FUNCTION_BLOCK bfb_offpeak_charging
  (* Standard: 61499-2 *)
  (* Version 0.1, 2018-00-09, palme, DESKTOP-TGOEKBD *)
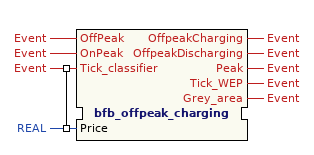
  EVENT_INPUT
    OffPeak;
    OnPeak;
    Tick_classifier WITH Price;
  END_EVENT
  EVENT_OUTPUT
    OffpeakCharging;
    OffpeakDischarging;
    Peak;
    Tick_WEP;
    Grey_area;
  END_EVENT
  VAR_INPUT
    Price : REAL;
  END_VAR
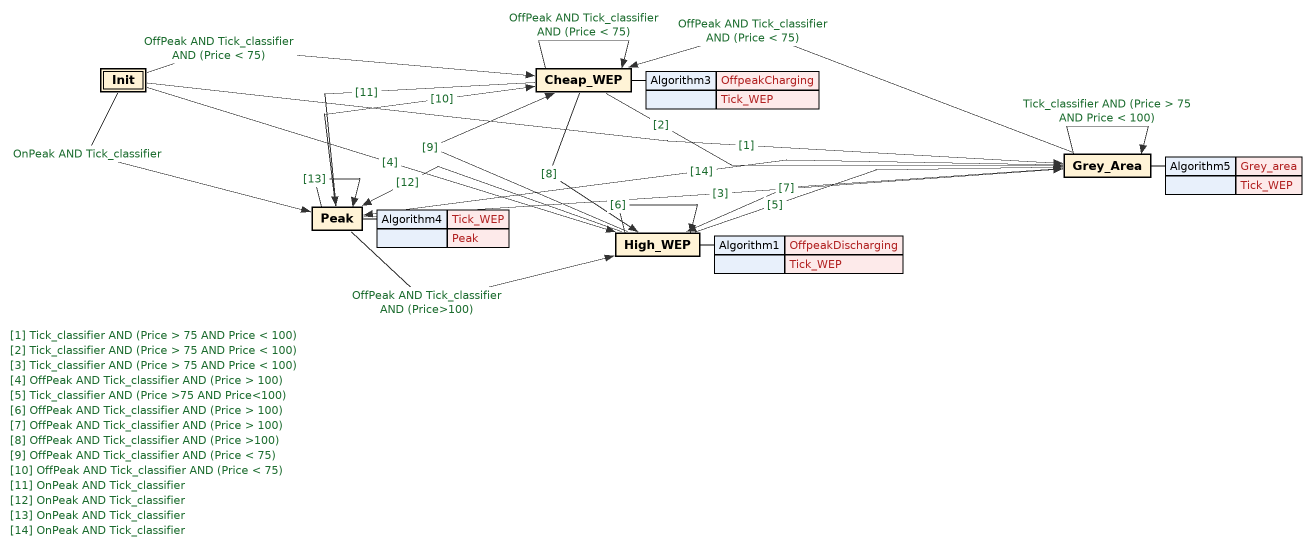
  EC_STATES
    Init;
    Cheap_WEP : Algorithm3 -> OffpeakCharging, -> Tick_WEP;
    High_WEP : Algorithm1 -> OffpeakDischarging, -> Tick_WEP;
    Peak : Algorithm4 -> Tick_WEP, -> Peak;
    Grey_Area : Algorithm5 -> Grey_area, -> Tick_WEP;
  END_STATES
  EC_TRANSITIONS
    Init TO Peak := OnPeak AND Tick_classifier;
    Init TO Grey_Area := Tick_classifier AND (Price > 75 AND Price < 100);
    Init TO Cheap_WEP := OffPeak AND Tick_classifier AND (Price < 75);
    Init TO High_WEP := OffPeak AND Tick_classifier AND (Price > 100);
    Cheap_WEP TO Peak := OnPeak AND Tick_classifier;
    Cheap_WEP TO Grey_Area := Tick_classifier AND (Price > 75 AND Price < 100);
    Cheap_WEP TO High_WEP := OffPeak AND Tick_classifier AND (Price >100);
    Cheap_WEP TO Cheap_WEP := OffPeak AND Tick_classifier AND (Price < 75);
    High_WEP TO Peak := OnPeak AND Tick_classifier;
    High_WEP TO Grey_Area := Tick_classifier AND (Price >75 AND Price<100);
    High_WEP TO Cheap_WEP := OffPeak AND Tick_classifier AND (Price < 75);
    High_WEP TO High_WEP := OffPeak AND Tick_classifier AND (Price > 100);
    Peak TO Peak := OnPeak AND Tick_classifier;
    Peak TO Grey_Area := Tick_classifier AND (Price > 75 AND Price < 100);
    Peak TO Cheap_WEP := OffPeak AND Tick_classifier AND (Price < 75);
    Peak TO High_WEP := OffPeak AND Tick_classifier AND (Price>100);
    Grey_Area TO Peak := OnPeak AND Tick_classifier;
    Grey_Area TO High_WEP := OffPeak AND Tick_classifier AND (Price > 100);
    Grey_Area TO Cheap_WEP := OffPeak AND Tick_classifier AND (Price < 75);
    Grey_Area TO Grey_Area := Tick_classifier AND (Price > 75 AND Price < 100);
  END_TRANSITIONS
  ALGORITHM Algorithm1 IN C:
printf("  High WEP   \r\n");
  END_ALGORITHM
  ALGORITHM Algorithm2 IN C:
printf(" No Charging..... \r\n ");
  END_ALGORITHM
  ALGORITHM Algorithm3 IN C:
printf("cheap WEP \r\n");
  END_ALGORITHM
  ALGORITHM Algorithm4 IN C:
printf("peak..... \r\n");
  END_ALGORITHM
  ALGORITHM Algorithm5 IN C:
printf("Grey Area");
  END_ALGORITHM
END_FUNCTION_BLOCK
